// TIA Portal project "plc_logging_siemens" (V17)

(* hardware
DEVICE "S7-1500/ET200MP station_1"  S7-1500 station
   slot 0: "Rail_0"  Rack  6ES7 590-1***0-0AA0
   slot 1: "PLC_1"  CPU 1511T-1 PN  6ES7 511-1TK01-0AB0  V2.9
      slot 3: "CPU display_1"  6ES7591-1AA00-0AA0
      slot 32768: "PROFINET interface_1"  X1
         slot 32769: "Port_1"  X1 P1
         slot 32770: "Port_2"  X1 P2
      slot 34817: "Virtual CP interface port_1"  Virtual CP interface port  Virtual CP interface port
*)

// ===== PLC "PLC_1"  CPU 1511T-1 PN =====

VAR_GLOBAL   // PLC tag table "Default tag table"
   "System_Byte" AT %MB1 : Byte;
   "FirstScan" AT %M1.0 : Bool;
   "DiagStatusUpdate" AT %M1.1 : Bool;
   "AlwaysTRUE" AT %M1.2 : Bool;
   "AlwaysFALSE" AT %M1.3 : Bool;
   "Clock_Byte" AT %MB0 : Byte;
   "Clock_10Hz" AT %M0.0 : Bool;
   "Clock_5Hz" AT %M0.1 : Bool;
   "Clock_2.5Hz" AT %M0.2 : Bool;
   "Clock_2Hz" AT %M0.3 : Bool;
   "Clock_1.25Hz" AT %M0.4 : Bool;
   "Clock_1Hz" AT %M0.5 : Bool;
   "Clock_0.625Hz" AT %M0.6 : Bool;
   "Clock_0.5Hz" AT %M0.7 : Bool;
END_VAR

DATA_BLOCK "test_logger_DB"   // DB2
{ S7_Optimized_Access := 'TRUE' }
VERSION : 0.1
// stored: InstanceOfName test_logger
"test_logger"
BEGIN
END_DATA_BLOCK

// folder: logger

DATA_BLOCK "logger"   // DB1
{ S7_Optimized_Access := 'TRUE' }
VERSION : 0.1
// stored: InstanceOfName LoggerFb
"LoggerFb"
BEGIN
END_DATA_BLOCK

DATA_BLOCK "LoggerLevels"   // DB3
{ S7_Optimized_Access := 'TRUE' }
VERSION : 0.1
   VAR
      NOTSET : USInt := 0;   // logging everything
      DEBUG : USInt := 10;
      INFO : USInt := 20;
      WARNING : USInt := 30;
      ERROR : USInt := 40;
      CRITICAL : USInt := 50;
      DISABLE : USInt := 100;   // logging disabled
   END_VAR
BEGIN
END_DATA_BLOCK

// folder: (top level)

FUNCTION_BLOCK "test_logger"   // FB2, SCL
{ S7_Optimized_Access := 'TRUE' }
VERSION : 0.1
   VAR
      prev : Struct
         clock : Bool;
      END_STRUCT;
   END_VAR
BEGIN
   "logger.config_in_block"(level := "LoggerLevels".DEBUG,
                            block_title := 'test_logger_block');


   if "Clock_0.5Hz" AND NOT #prev.clock THEN
       "logger.debug_3"(msg := 'test debug message, SP: {0}, PV: {1}, add: {2}',
                        value_0 := REAL_TO_STRING(10),
                        value_1 := REAL_TO_STRING(11),
                        value_2 := REAL_TO_STRING(12)
       );
       //"logger.info_0"('test info message');
       //"logger.warning_0"('test warning message');
       //"logger.error_0"('test error message');
       //"logger.critical_0"(msg := 'test critical message');
   END_IF;

   #prev.clock := "Clock_0.5Hz";
END_FUNCTION_BLOCK

ORGANIZATION_BLOCK "Main"   // OB1, SCL, ProgramCycle
TITLE = "Main Program Sweep (Cycle)"
{ S7_Optimized_Access := 'TRUE' }
VERSION : 0.1
   VAR_INPUT
      Initial_Call : Bool;   // Initial call of this OB
      Remanence : Bool;   // =True, if remanent data are available
   END_VAR
BEGIN
   "test_logger_DB"();


   "logger"(global_logger_level := "LoggerLevels".DEBUG,
            ip_1 := 10,
            ip_2 := 101,
            ip_3 := 50,
            ip_4 := 17,
            port_number := 8000,
            interface_id := "Local~PROFINET_interface_1"
   );
END_ORGANIZATION_BLOCK

// folder: logger

FUNCTION_BLOCK "LoggerFb"   // FB1, SCL
{ S7_Optimized_Access := 'TRUE' }
VERSION : 0.1
   VAR_INPUT
      global_logger_level : USInt := 0;   // Filter all logging messages
      ip_1 : USInt := 192;
      ip_2 : USInt := 168;
      ip_3 : USInt := 10;
      ip_4 : USInt := 2;
      port_number : UInt := 4567;
      interface_id : UInt := 64;
   END_VAR
   VAR_OUTPUT
      buffer_size : Int;
   END_VAR
   VAR
      prev : Struct
         state : Int;
      END_STRUCT;
      diag : Struct
         tcon_done_counter : UDInt;
         tcon_error_counter : UDInt;
         tcon_error_status : Word;
         timeout_counter : UDInt;
         tsend_done_counter : UDInt;
         tsend_error_counter : UDInt;
         tsend_error_status : Word;
      END_STRUCT;
      connect : TCON_IP_v4;
      data : String;
      buffer : Array[0..9] of String;
      state : Int;
      timeout : TON_TIME;
      init : Bool := TRUE;   // TRUE = initialize function block
      config_in_block : Struct
         level : USInt;
         block_title : String;
      END_STRUCT;
      tcon : TCON;
      tsend : TSEND;
      tdiscon : TDISCON;
      connect_id : Conn_Ouc := 16#0001;
   END_VAR
   VAR_TEMP
      i : Int;
      com_rst : Bool;
   END_VAR
   VAR CONSTANT
      BUFFER_SIZE_ : Int := 9;
      ST_STOP : Int;
      ST_CONNECT : Int := 1;
      ST_WAIT : Int := 2;
      ST_SEND : Int := 3;
      ST_DISCON : Int := 4;
   END_VAR
BEGIN
   (*Блок логгера.*)

   // -----------------------------------------------------------------------------

   if #init THEN
       // first execution
       #connect.RemoteAddress.ADDR[1] := #ip_1;
       #connect.RemoteAddress.ADDR[2] := #ip_2;
       #connect.RemoteAddress.ADDR[3] := #ip_3;
       #connect.RemoteAddress.ADDR[4] := #ip_4;
       #connect.RemotePort := #port_number;
       #connect.LocalPort := #port_number;
       #connect.ActiveEstablished := true;
       #connect.InterfaceId := #interface_id;
       //#connect.ID := #id;
       #state := #ST_STOP;
       #connect.ConnectionType := 11;

       #buffer_size := #"BUFFER_SIZE_";
   END_IF;

   case #state OF
       #ST_STOP:
           if #global_logger_level < "LoggerLevels".DISABLE THEN
               #state := #ST_CONNECT;
               for #i := 0 TO #"BUFFER_SIZE_" DO
                   #buffer[#i] := '';
               END_FOR;
           END_IF;

       #ST_CONNECT:
           if #global_logger_level = "LoggerLevels".DISABLE OR #init THEN
               #state := #ST_STOP;
           ELSIF #tcon.DONE THEN
               // done
               #diag.tcon_done_counter += 1;
               #state := #ST_WAIT;
           ELSIF #tcon.ERROR THEN
               // error
               #diag.tcon_error_counter += 1;
               #diag.tcon_error_status := #tcon.STATUS;
               #state := #ST_STOP;
               if #tcon.STATUS = 16#80A3 THEN
                   #connect_id += 1;
               END_IF;
           ELSIF #timeout.Q THEN
               // timeout
               #diag.timeout_counter += 1;
               #state := #ST_STOP;
           END_IF;

       #ST_WAIT:
           if #global_logger_level = "LoggerLevels".DISABLE OR #init THEN
               #state := #ST_DISCON;
           END_IF;

           if #buffer[0] <> '' THEN
               #data := #buffer[0];
               for #i := 0 TO #"BUFFER_SIZE_" - 1 DO
                   #buffer[#i] := #buffer[#i + 1];
               END_FOR;
               #buffer[#"BUFFER_SIZE_"] := '';
               #state := #ST_SEND;
           END_IF;

       #ST_SEND:
           if #global_logger_level = "LoggerLevels".DISABLE OR #init THEN
               #state := #ST_DISCON;
           ELSIF #tsend.DONE THEN
               // done
               #diag.tsend_done_counter += 1;
               #state := #ST_WAIT;
           ELSIF #tsend.ERROR THEN
               // error
               #diag.tsend_error_counter += 1;
               #diag.tsend_error_status := #tsend.STATUS;
               #state := #ST_DISCON;
           ELSIF #timeout.Q THEN
               // timeout
               #diag.timeout_counter += 1;
               #state := #ST_DISCON;
           END_IF;

       #ST_DISCON:
           if #tdiscon.DONE OR #tdiscon.ERROR OR #timeout.Q THEN
               #state := #ST_STOP;
           END_IF;

   END_CASE;

   #timeout(IN := #state = #prev.state,
            PT := T#5s);

   #connect.ID := #connect_id;
   #tcon(REQ := #state = #ST_CONNECT,
         ID := #connect_id,
         CONNECT := #connect);

   #tsend(REQ := #state = #ST_SEND,
          ID := #connect_id,
          LEN := INT_TO_UDINT(LEN(#data)) + 2, // why 2 ???
          DATA := #data);

   #tdiscon(REQ := #state = #ST_DISCON,
            ID := #connect_id);

   #init := false;
   #prev.state := #state;
END_FUNCTION_BLOCK

FUNCTION "logger.debug_1" : Void   // FC1, SCL
{ S7_Optimized_Access := 'TRUE' }
VERSION : 0.1
   VAR_INPUT
      msg : String;   // message for logging
      value_0 : String;   // additional value 0
   END_VAR
   VAR_TEMP
      str : String;
   END_VAR
BEGIN
   IF MAX_USINT(IN1 := "logger".config_in_block.level, IN2 := "logger".global_logger_level) >
       "LoggerLevels".DEBUG THEN
       RETURN;
   END_IF;

   #str := '';
   #str := CONCAT_STRING(IN1 := #str, IN2 := #msg);
   #str := CONCAT_STRING(IN1 := #str, IN2 := '$t');
   #str := CONCAT_STRING(IN1 := #str, IN2 := #value_0);

   "logger._log"(level := "LoggerLevels".DEBUG,
                 msg := #str
   );
END_FUNCTION

FUNCTION "logger._log" : Void   // FC2, SCL
{ S7_Optimized_Access := 'TRUE' }
VERSION : 0.1
   VAR_INPUT
      level : USInt;
      msg : String;
   END_VAR
   VAR_TEMP
      temp_dtl : DTL;
      temp_int : Int;
      ts : String;
      pos : UInt;
      i : Int;
      str : String;
   END_VAR
BEGIN
   (*Add message to buffer.
   Format: LEVEL, TIMESTAMP, BLOCK_TITLE, MESSAGE
   Separator - \t.
   *)

   REGION timestamp
       // timestamp
       #temp_int := RD_LOC_T(#temp_dtl);

       #ts := 'YYYY-MM-DD HH:MM:SS,NNNNNNNNN';
       #pos := 1;
       VAL_STRG(IN := #temp_dtl.YEAR,
                SIZE := 4,
                PREC := 0,
                FORMAT := 0,
                P := #pos,
                OUT => #ts);
       #pos := 6;
       VAL_STRG(IN := #temp_dtl.MONTH,
                SIZE := 2,
                PREC := 0,
                FORMAT := 0,
                P := #pos,
                OUT => #ts);
       #pos := 9;
       VAL_STRG(IN := #temp_dtl.DAY,
                SIZE := 2,
                PREC := 0,
                FORMAT := 0,
                P := #pos,
                OUT => #ts);
       #pos := 12;
       VAL_STRG(IN := #temp_dtl.HOUR,
                SIZE := 2,
                PREC := 0,
                FORMAT := 0,
                P := #pos,
                OUT => #ts);
       #pos := 15;
       VAL_STRG(IN := #temp_dtl.MINUTE,
                SIZE := 2,
                PREC := 0,
                FORMAT := 0,
                P := #pos,
                OUT => #ts);
       #pos := 18;
       VAL_STRG(IN := #temp_dtl.SECOND,
                SIZE := 2,
                PREC := 0,
                FORMAT := 0,
                P := #pos,
                OUT => #ts);
       #pos := 21;
       VAL_STRG(IN := #temp_dtl.NANOSECOND,
                SIZE := 0,
                PREC := 0,
                FORMAT := 0,
                P := #pos,
                OUT => #ts);
       FOR #i := 1 TO LEN(#ts) DO
           // fill with zeros
           IF #ts[#i] = ' ' THEN
               #ts[#i] := '0';
           END_IF;
       END_FOR;
       #ts[11] := ' '; // separator between day and hours
   END_REGION

   #str := '';
   #str := CONCAT_STRING(IN1 := #str, IN2 := USINT_TO_STRING(#level));
   #str := CONCAT_STRING(IN1 := #str, IN2 := '$t');
   #str := CONCAT_STRING(IN1 := #str, IN2 := #ts);
   #str := CONCAT_STRING(IN1 := #str, IN2 := '$t');
   #str := CONCAT_STRING(IN1 := #str, IN2 := "logger".config_in_block.block_title);
   #str := CONCAT_STRING(IN1 := #str, IN2 := '$t');
   #str := CONCAT_STRING(IN1 := #str, IN2 := #msg);
   #str := CONCAT_STRING(IN1 := #str, IN2 := '$r');

   FOR #i := 0 TO "logger".buffer_size DO
       IF "logger".buffer[#i] = '' THEN
           "logger".buffer[#i] := #str;
           RETURN;
       END_IF;
   END_FOR;
END_FUNCTION

FUNCTION "logger.debug_0" : Void   // FC3, SCL
{ S7_Optimized_Access := 'TRUE' }
VERSION : 0.1
   VAR_INPUT
      msg : String;   // message for logging
   END_VAR
BEGIN
   IF MAX_USINT(IN1 := "logger".config_in_block.level, IN2 := "logger".global_logger_level) >
       "LoggerLevels".DEBUG THEN
       RETURN;
   END_IF;

   "logger._log"(level := "LoggerLevels".DEBUG,
                 msg := #msg
   );
END_FUNCTION

FUNCTION "logger.info_0" : Void   // FC4, SCL
{ S7_Optimized_Access := 'TRUE' }
VERSION : 0.1
   VAR_INPUT
      msg : String;   // message for logging
   END_VAR
BEGIN
   IF MAX_USINT(IN1 := "logger".config_in_block.level, IN2 := "logger".global_logger_level) >
       "LoggerLevels".INFO THEN
       RETURN;
   END_IF;

   "logger._log"(level := "LoggerLevels".INFO,
                 msg := #msg
   );
END_FUNCTION

FUNCTION "logger.config_in_block" : Void   // FC5, SCL
{ S7_Optimized_Access := 'TRUE' }
VERSION : 0.1
   VAR_INPUT
      level : USInt;
      block_title : String;
   END_VAR
BEGIN
   "logger".config_in_block.block_title := #block_title;
   "logger".config_in_block.level := #level;
END_FUNCTION

FUNCTION "logger.warning_0" : Void   // FC6, SCL
{ S7_Optimized_Access := 'TRUE' }
VERSION : 0.1
   VAR_INPUT
      msg : String;   // message for logging
   END_VAR
BEGIN
   IF MAX_USINT(IN1 := "logger".config_in_block.level, IN2 := "logger".global_logger_level) >
       "LoggerLevels".WARNING THEN
       RETURN;
   END_IF;

   "logger._log"(level := "LoggerLevels".WARNING,
                 msg := #msg
   );
END_FUNCTION

FUNCTION "logger.error_0" : Void   // FC7, SCL
{ S7_Optimized_Access := 'TRUE' }
VERSION : 0.1
   VAR_INPUT
      msg : String;   // message for logging
   END_VAR
BEGIN
   IF MAX_USINT(IN1 := "logger".config_in_block.level, IN2 := "logger".global_logger_level) >
       "LoggerLevels".ERROR THEN
       RETURN;
   END_IF;

   "logger._log"(level := "LoggerLevels".ERROR,
                 msg := #msg
   );
END_FUNCTION

FUNCTION "logger.critical_0" : Void   // FC8, SCL
{ S7_Optimized_Access := 'TRUE' }
VERSION : 0.1
   VAR_INPUT
      msg : String;   // message for logging
   END_VAR
BEGIN
   IF MAX_USINT(IN1 := "logger".config_in_block.level, IN2 := "logger".global_logger_level) >
       "LoggerLevels".CRITICAL THEN
       RETURN;
   END_IF;

   "logger._log"(level := "LoggerLevels".CRITICAL,
                 msg := #msg
   );
END_FUNCTION

FUNCTION "logger.debug_2" : Void   // FC9, SCL
{ S7_Optimized_Access := 'TRUE' }
VERSION : 0.1
   VAR_INPUT
      msg : String;   // message for logging
      value_0 : String;   // additional value 0
      value_1 : String;   // additional value 1
   END_VAR
   VAR_TEMP
      str : String;
   END_VAR
BEGIN
   IF MAX_USINT(IN1 := "logger".config_in_block.level, IN2 := "logger".global_logger_level) >
       "LoggerLevels".DEBUG THEN
       RETURN;
   END_IF;

   #str := '';
   #str := CONCAT_STRING(IN1 := #str, IN2 := #msg);
   #str := CONCAT_STRING(IN1 := #str, IN2 := '$t');
   #str := CONCAT_STRING(IN1 := #str, IN2 := #value_0);
   #str := CONCAT_STRING(IN1 := #str, IN2 := '$t');
   #str := CONCAT_STRING(IN1 := #str, IN2 := #value_1);

   "logger._log"(level := "LoggerLevels".DEBUG,
                 msg := #str
   );
END_FUNCTION

FUNCTION "logger.debug_3" : Void   // FC10, SCL
{ S7_Optimized_Access := 'TRUE' }
VERSION : 0.1
   VAR_INPUT
      msg : String;   // message for logging
      value_0 : String;   // additional value 0
      value_1 : String;   // additional value 1
      value_2 : String;   // additional value 2
   END_VAR
   VAR_TEMP
      str : String;
   END_VAR
BEGIN
   IF MAX_USINT(IN1 := "logger".config_in_block.level, IN2 := "logger".global_logger_level) >
       "LoggerLevels".DEBUG THEN
       RETURN;
   END_IF;

   #str := '';
   #str := CONCAT_STRING(IN1 := #str, IN2 := #msg);
   #str := CONCAT_STRING(IN1 := #str, IN2 := '$t');
   #str := CONCAT_STRING(IN1 := #str, IN2 := #value_0);
   #str := CONCAT_STRING(IN1 := #str, IN2 := '$t');
   #str := CONCAT_STRING(IN1 := #str, IN2 := #value_1);
   #str := CONCAT_STRING(IN1 := #str, IN2 := '$t');
   #str := CONCAT_STRING(IN1 := #str, IN2 := #value_2);

   "logger._log"(level := "LoggerLevels".DEBUG,
                 msg := #str
   );
END_FUNCTION

FUNCTION "logger.info_1" : Void   // FC11, SCL
{ S7_Optimized_Access := 'TRUE' }
VERSION : 0.1
   VAR_INPUT
      msg : String;   // message for logging
      value_0 : String;   // additional value 0
   END_VAR
   VAR_TEMP
      str : String;
   END_VAR
BEGIN
   IF MAX_USINT(IN1 := "logger".config_in_block.level, IN2 := "logger".global_logger_level) >
       "LoggerLevels".INFO THEN
       RETURN;
   END_IF;

   #str := '';
   #str := CONCAT_STRING(IN1 := #str, IN2 := #msg);
   #str := CONCAT_STRING(IN1 := #str, IN2 := '$t');
   #str := CONCAT_STRING(IN1 := #str, IN2 := #value_0);

   "logger._log"(level := "LoggerLevels".INFO,
                 msg := #str
   );
END_FUNCTION

FUNCTION "logger.error_1" : Void   // FC12, SCL
{ S7_Optimized_Access := 'TRUE' }
VERSION : 0.1
   VAR_INPUT
      msg : String;   // message for logging
      value_0 : String;   // additional value 0
   END_VAR
   VAR_TEMP
      str : String;
   END_VAR
BEGIN
   IF MAX_USINT(IN1 := "logger".config_in_block.level, IN2 := "logger".global_logger_level) >
       "LoggerLevels".ERROR THEN
       RETURN;
   END_IF;

   #str := '';
   #str := CONCAT_STRING(IN1 := #str, IN2 := #msg);
   #str := CONCAT_STRING(IN1 := #str, IN2 := '$t');
   #str := CONCAT_STRING(IN1 := #str, IN2 := #value_0);

   "logger._log"(level := "LoggerLevels".ERROR,
                 msg := #str
   );
END_FUNCTION

FUNCTION "logger.critical_1" : Void   // FC13, SCL
{ S7_Optimized_Access := 'TRUE' }
VERSION : 0.1
   VAR_INPUT
      msg : String;   // message for logging
      value_0 : String;   // additional value 0
   END_VAR
   VAR_TEMP
      str : String;
   END_VAR
BEGIN
   IF MAX_USINT(IN1 := "logger".config_in_block.level, IN2 := "logger".global_logger_level) >
       "LoggerLevels".CRITICAL THEN
       RETURN;
   END_IF;

   #str := '';
   #str := CONCAT_STRING(IN1 := #str, IN2 := #msg);
   #str := CONCAT_STRING(IN1 := #str, IN2 := '$t');
   #str := CONCAT_STRING(IN1 := #str, IN2 := #value_0);

   "logger._log"(level := "LoggerLevels".CRITICAL,
                 msg := #str
   );
END_FUNCTION

FUNCTION "logger.warning_1" : Void   // FC14, SCL
{ S7_Optimized_Access := 'TRUE' }
VERSION : 0.1
   VAR_INPUT
      msg : String;   // message for logging
      value_0 : String;   // additional value 0
   END_VAR
   VAR_TEMP
      str : String;
   END_VAR
BEGIN
   IF MAX_USINT(IN1 := "logger".config_in_block.level, IN2 := "logger".global_logger_level) >
       "LoggerLevels".WARNING THEN
       RETURN;
   END_IF;

   #str := '';
   #str := CONCAT_STRING(IN1 := #str, IN2 := #msg);
   #str := CONCAT_STRING(IN1 := #str, IN2 := '$t');
   #str := CONCAT_STRING(IN1 := #str, IN2 := #value_0);

   "logger._log"(level := "LoggerLevels".WARNING,
                 msg := #str
   );
END_FUNCTION

FUNCTION "logger.warning_2" : Void   // FC15, SCL
{ S7_Optimized_Access := 'TRUE' }
VERSION : 0.1
   VAR_INPUT
      msg : String;   // message for logging
      value_0 : String;   // additional value 0
      value_1 : String;   // additional value 1
   END_VAR
   VAR_TEMP
      str : String;
   END_VAR
BEGIN
   IF MAX_USINT(IN1 := "logger".config_in_block.level, IN2 := "logger".global_logger_level) >
       "LoggerLevels".WARNING THEN
       RETURN;
   END_IF;

   #str := '';
   #str := CONCAT_STRING(IN1 := #str, IN2 := #msg);
   #str := CONCAT_STRING(IN1 := #str, IN2 := '$t');
   #str := CONCAT_STRING(IN1 := #str, IN2 := #value_0);
   #str := CONCAT_STRING(IN1 := #str, IN2 := '$t');
   #str := CONCAT_STRING(IN1 := #str, IN2 := #value_1);

   "logger._log"(level := "LoggerLevels".WARNING,
                 msg := #str
   );
END_FUNCTION

FUNCTION "logger.info_2" : Void   // FC16, SCL
{ S7_Optimized_Access := 'TRUE' }
VERSION : 0.1
   VAR_INPUT
      msg : String;   // message for logging
      value_0 : String;   // additional value 0
      value_1 : String;   // additional value 1
   END_VAR
   VAR_TEMP
      str : String;
   END_VAR
BEGIN
   IF MAX_USINT(IN1 := "logger".config_in_block.level, IN2 := "logger".global_logger_level) >
       "LoggerLevels".INFO THEN
       RETURN;
   END_IF;

   #str := '';
   #str := CONCAT_STRING(IN1 := #str, IN2 := #msg);
   #str := CONCAT_STRING(IN1 := #str, IN2 := '$t');
   #str := CONCAT_STRING(IN1 := #str, IN2 := #value_0);
   #str := CONCAT_STRING(IN1 := #str, IN2 := '$t');
   #str := CONCAT_STRING(IN1 := #str, IN2 := #value_1);

   "logger._log"(level := "LoggerLevels".INFO,
                 msg := #str
   );
END_FUNCTION

FUNCTION "logger.critical_2" : Void   // FC17, SCL
{ S7_Optimized_Access := 'TRUE' }
VERSION : 0.1
   VAR_INPUT
      msg : String;   // message for logging
      value_0 : String;   // additional value 0
      value_1 : String;   // additional value 1
   END_VAR
   VAR_TEMP
      str : String;
   END_VAR
BEGIN
   IF MAX_USINT(IN1 := "logger".config_in_block.level, IN2 := "logger".global_logger_level) >
       "LoggerLevels".CRITICAL THEN
       RETURN;
   END_IF;

   #str := '';
   #str := CONCAT_STRING(IN1 := #str, IN2 := #msg);
   #str := CONCAT_STRING(IN1 := #str, IN2 := '$t');
   #str := CONCAT_STRING(IN1 := #str, IN2 := #value_0);
   #str := CONCAT_STRING(IN1 := #str, IN2 := '$t');
   #str := CONCAT_STRING(IN1 := #str, IN2 := #value_1);

   "logger._log"(level := "LoggerLevels".CRITICAL,
                 msg := #str
   );
END_FUNCTION

FUNCTION "logger.error_2" : Void   // FC18, SCL
{ S7_Optimized_Access := 'TRUE' }
VERSION : 0.1
   VAR_INPUT
      msg : String;   // message for logging
      value_0 : String;   // additional value 0
      value_1 : String;   // additional value 1
   END_VAR
   VAR_TEMP
      str : String;
   END_VAR
BEGIN
   IF MAX_USINT(IN1 := "logger".config_in_block.level, IN2 := "logger".global_logger_level) >
       "LoggerLevels".ERROR THEN
       RETURN;
   END_IF;

   #str := '';
   #str := CONCAT_STRING(IN1 := #str, IN2 := #msg);
   #str := CONCAT_STRING(IN1 := #str, IN2 := '$t');
   #str := CONCAT_STRING(IN1 := #str, IN2 := #value_0);
   #str := CONCAT_STRING(IN1 := #str, IN2 := '$t');
   #str := CONCAT_STRING(IN1 := #str, IN2 := #value_1);

   "logger._log"(level := "LoggerLevels".ERROR,
                 msg := #str
   );
END_FUNCTION

FUNCTION "logger.error_3" : Void   // FC19, SCL
{ S7_Optimized_Access := 'TRUE' }
VERSION : 0.1
   VAR_INPUT
      msg : String;   // message for logging
      value_0 : String;   // additional value 0
      value_1 : String;   // additional value 1
      value_2 : String;   // additional value 2
   END_VAR
   VAR_TEMP
      str : String;
   END_VAR
BEGIN
   IF MAX_USINT(IN1 := "logger".config_in_block.level, IN2 := "logger".global_logger_level) >
       "LoggerLevels".ERROR THEN
       RETURN;
   END_IF;

   #str := '';
   #str := CONCAT_STRING(IN1 := #str, IN2 := #msg);
   #str := CONCAT_STRING(IN1 := #str, IN2 := '$t');
   #str := CONCAT_STRING(IN1 := #str, IN2 := #value_0);
   #str := CONCAT_STRING(IN1 := #str, IN2 := '$t');
   #str := CONCAT_STRING(IN1 := #str, IN2 := #value_1);
   #str := CONCAT_STRING(IN1 := #str, IN2 := '$t');
   #str := CONCAT_STRING(IN1 := #str, IN2 := #value_2);

   "logger._log"(level := "LoggerLevels".ERROR,
                 msg := #str
   );
END_FUNCTION

FUNCTION "logger.info_3" : Void   // FC20, SCL
{ S7_Optimized_Access := 'TRUE' }
VERSION : 0.1
   VAR_INPUT
      msg : String;   // message for logging
      value_0 : String;   // additional value 0
      value_1 : String;   // additional value 1
      value_2 : String;   // additional value 2
   END_VAR
   VAR_TEMP
      str : String;
   END_VAR
BEGIN
   IF MAX_USINT(IN1 := "logger".config_in_block.level, IN2 := "logger".global_logger_level) >
       "LoggerLevels".INFO THEN
       RETURN;
   END_IF;

   #str := '';
   #str := CONCAT_STRING(IN1 := #str, IN2 := #msg);
   #str := CONCAT_STRING(IN1 := #str, IN2 := '$t');
   #str := CONCAT_STRING(IN1 := #str, IN2 := #value_0);
   #str := CONCAT_STRING(IN1 := #str, IN2 := '$t');
   #str := CONCAT_STRING(IN1 := #str, IN2 := #value_1);
   #str := CONCAT_STRING(IN1 := #str, IN2 := '$t');
   #str := CONCAT_STRING(IN1 := #str, IN2 := #value_2);

   "logger._log"(level := "LoggerLevels".INFO,
                 msg := #str
   );
END_FUNCTION

FUNCTION "logger.critical_3" : Void   // FC21, SCL
{ S7_Optimized_Access := 'TRUE' }
VERSION : 0.1
   VAR_INPUT
      msg : String;   // message for logging
      value_0 : String;   // additional value 0
      value_1 : String;   // additional value 1
      value_2 : String;   // additional value 2
   END_VAR
   VAR_TEMP
      str : String;
   END_VAR
BEGIN
   IF MAX_USINT(IN1 := "logger".config_in_block.level, IN2 := "logger".global_logger_level) >
       "LoggerLevels".CRITICAL THEN
       RETURN;
   END_IF;

   #str := '';
   #str := CONCAT_STRING(IN1 := #str, IN2 := #msg);
   #str := CONCAT_STRING(IN1 := #str, IN2 := '$t');
   #str := CONCAT_STRING(IN1 := #str, IN2 := #value_0);
   #str := CONCAT_STRING(IN1 := #str, IN2 := '$t');
   #str := CONCAT_STRING(IN1 := #str, IN2 := #value_1);
   #str := CONCAT_STRING(IN1 := #str, IN2 := '$t');
   #str := CONCAT_STRING(IN1 := #str, IN2 := #value_2);

   "logger._log"(level := "LoggerLevels".CRITICAL,
                 msg := #str
   );
END_FUNCTION

FUNCTION "logger.warning_3" : Void   // FC22, SCL
{ S7_Optimized_Access := 'TRUE' }
VERSION : 0.1
   VAR_INPUT
      msg : String;   // message for logging
      value_0 : String;   // additional value 0
      value_1 : String;   // additional value 1
      value_2 : String;   // additional value 2
   END_VAR
   VAR_TEMP
      str : String;
   END_VAR
BEGIN
   IF MAX_USINT(IN1 := "logger".config_in_block.level, IN2 := "logger".global_logger_level) >
       "LoggerLevels".WARNING THEN
       RETURN;
   END_IF;

   #str := '';
   #str := CONCAT_STRING(IN1 := #str, IN2 := #msg);
   #str := CONCAT_STRING(IN1 := #str, IN2 := '$t');
   #str := CONCAT_STRING(IN1 := #str, IN2 := #value_0);
   #str := CONCAT_STRING(IN1 := #str, IN2 := '$t');
   #str := CONCAT_STRING(IN1 := #str, IN2 := #value_1);
   #str := CONCAT_STRING(IN1 := #str, IN2 := '$t');
   #str := CONCAT_STRING(IN1 := #str, IN2 := #value_2);

   "logger._log"(level := "LoggerLevels".WARNING,
                 msg := #str
   );
END_FUNCTION

// ===== library: MasterCopy "Copy of Program blocks in logger" =====

// folder: logger

DATA_BLOCK "logger"   // DB1
{ S7_Optimized_Access := 'TRUE' }
VERSION : 0.1
// stored: InstanceOfName LoggerFb
"LoggerFb"
BEGIN
END_DATA_BLOCK

DATA_BLOCK "LoggerLevels"   // DB3
{ S7_Optimized_Access := 'TRUE' }
VERSION : 0.1
   VAR
      NOTSET : USInt := 0;   // logging everything
      DEBUG : USInt := 10;
      INFO : USInt := 20;
      WARNING : USInt := 30;
      ERROR : USInt := 40;
      CRITICAL : USInt := 50;
      DISABLE : USInt := 100;   // logging disabled
   END_VAR
BEGIN
END_DATA_BLOCK

FUNCTION_BLOCK "LoggerFb"   // FB1, SCL
{ S7_Optimized_Access := 'TRUE' }
VERSION : 0.1
   VAR_INPUT
      global_logger_level : USInt := 0;   // Filter all logging messages
      ip_1 : USInt := 10;
      ip_2 : USInt := 101;
      ip_3 : USInt := 50;
      ip_4 : USInt := 17;
      port_number : UInt := 4567;
      interface_id : UInt := 64;
      id : Conn_Ouc := 1;
   END_VAR
   VAR_OUTPUT
      buffer_size : Int;
   END_VAR
   VAR
      tsend : TSEND_C;
      connect : TCON_IP_v4;
      data : String;
      buffer : Array[0..9] of String;
      state : Int;
      timeout : TON_TIME;
      init : Bool := TRUE;   // TRUE = initialize function block
      config_in_block : Struct
         level : USInt;
         block_title : String;
      END_STRUCT;
   END_VAR
   VAR_TEMP
      i : Int;
   END_VAR
   VAR CONSTANT
      ST_STOP : Int;
      ST_WAIT : Int := 1;
      ST_SEND : Int := 2;
      BUFFER_SIZE_ : Int := 9;
   END_VAR
BEGIN
   (*Блок логгера.*)

   // -----------------------------------------------------------------------------

   if #init THEN
       // first execution
       #init := false;
       #connect.RemoteAddress.ADDR[1] := #ip_1;
       #connect.RemoteAddress.ADDR[2] := #ip_2;
       #connect.RemoteAddress.ADDR[3] := #ip_3;
       #connect.RemoteAddress.ADDR[4] := #ip_4;
       #connect.RemotePort := #port_number;
       #connect.LocalPort := #port_number;
       #connect.ActiveEstablished := true;
       #connect.InterfaceId := #interface_id;
       #connect.ID := #id;
       #state := #ST_STOP;
       #connect.ConnectionType := 11;

       #buffer_size := #"BUFFER_SIZE_";
   END_IF;


   case #state OF
       #ST_STOP:
           if #global_logger_level < "LoggerLevels".DISABLE THEN
               #state := #ST_WAIT;
               for #i := 0 TO #"BUFFER_SIZE_" DO
                   #buffer[#i] := '';
               END_FOR;
           END_IF;

       #ST_WAIT:
           if #global_logger_level = "LoggerLevels".DISABLE THEN
               #state := #ST_STOP;
           END_IF;

           if #buffer[0] <> '' THEN
               #data := #buffer[0];
               for #i := 0 TO #"BUFFER_SIZE_" - 1 DO
                   #buffer[#i] := #buffer[#i + 1];
               END_FOR;
               #buffer[#"BUFFER_SIZE_"] := '';
               #state := #ST_SEND;
           END_IF;

       #ST_SEND:
           if #global_logger_level = "LoggerLevels".DISABLE THEN
               #state := #ST_STOP;
           ELSIF #tsend.DONE OR #tsend.ERROR OR #timeout.Q THEN
               #data := '';
               #state := #ST_WAIT;
           END_IF;

   END_CASE;

   #timeout(IN := #state = #ST_SEND,
            PT := T#30s);


   #tsend(REQ := #state = #ST_SEND,
          CONT := #state = #ST_SEND,
          CONNECT := #connect,
          DATA := #data
   );
END_FUNCTION_BLOCK

FUNCTION "logger.debug_1" : Void   // FC1, SCL
{ S7_Optimized_Access := 'TRUE' }
VERSION : 0.1
   VAR_INPUT
      msg : String;   // message for logging
      value_0 : String;   // additional value 0
   END_VAR
   VAR_TEMP
      str : String;
   END_VAR
BEGIN
   if "logger".config_in_block.level > "LoggerLevels".DEBUG THEN
       return;
   END_IF;

   #str := '';
   #str := CONCAT_STRING(IN1 := #str, IN2 := #msg);
   #str := CONCAT_STRING(IN1 := #str, IN2 := '$t');
   #str := CONCAT_STRING(IN1 := #str, IN2 := #value_0);

   "logger._log"(level := "LoggerLevels".DEBUG,
                 msg := #str
   );
END_FUNCTION

FUNCTION "logger._log" : Void   // FC2, SCL
{ S7_Optimized_Access := 'TRUE' }
VERSION : 0.1
   VAR_INPUT
      level : USInt;
      msg : String;
   END_VAR
   VAR_TEMP
      temp_dtl : DTL;
      temp_int : Int;
      ts : String;
      pos : UInt;
      i : Int;
      str : String;
   END_VAR
BEGIN
   (*Add message to buffer.
   Format: LEVEL, TIMESTAMP, BLOCK_TITLE, MESSAGE
   Separator - \t.
   *)

   region timestamp
       // timestamp
       #temp_int := RD_LOC_T(#temp_dtl);

       #ts := 'YYYY-MM-DD HH:MM:SS,NNNNNNNNN';
       #pos := 1;
       VAL_STRG(IN := #temp_dtl.YEAR,
                SIZE := 4,
                PREC := 0,
                FORMAT := 0,
                P := #pos,
                OUT => #ts);
       #pos := 6;
       VAL_STRG(IN := #temp_dtl.MONTH,
                SIZE := 2,
                PREC := 0,
                FORMAT := 0,
                P := #pos,
                OUT => #ts);
       #pos := 9;
       VAL_STRG(IN := #temp_dtl.DAY,
                SIZE := 2,
                PREC := 0,
                FORMAT := 0,
                P := #pos,
                OUT => #ts);
       #pos := 12;
       VAL_STRG(IN := #temp_dtl.HOUR,
                SIZE := 2,
                PREC := 0,
                FORMAT := 0,
                P := #pos,
                OUT => #ts);
       #pos := 15;
       VAL_STRG(IN := #temp_dtl.MINUTE,
                SIZE := 2,
                PREC := 0,
                FORMAT := 0,
                P := #pos,
                OUT => #ts);
       #pos := 18;
       VAL_STRG(IN := #temp_dtl.SECOND,
                SIZE := 2,
                PREC := 0,
                FORMAT := 0,
                P := #pos,
                OUT => #ts);
       #pos := 21;
       VAL_STRG(IN := #temp_dtl.NANOSECOND,
                SIZE := 0,
                PREC := 0,
                FORMAT := 0,
                P := #pos,
                OUT => #ts);
       for #i := 1 TO LEN(#ts) DO
           // fill with zeros
           if #ts[#i] = ' ' THEN
               #ts[#i] := '0';
           END_IF;
       END_FOR;
       #ts[11] := ' '; // separator between day and hours
   END_REGION

   #str := '';
   #str := CONCAT_STRING(IN1 := #str, IN2 := USINT_TO_STRING(#level));
   #str := CONCAT_STRING(IN1 := #str, IN2 := '$t');
   #str := CONCAT_STRING(IN1 := #str, IN2 := #ts);
   #str := CONCAT_STRING(IN1 := #str, IN2 := '$t');
   #str := CONCAT_STRING(IN1 := #str, IN2 := "logger".config_in_block.block_title);
   #str := CONCAT_STRING(IN1 := #str, IN2 := '$t');
   #str := CONCAT_STRING(IN1 := #str, IN2 := #msg);

   for #i := 0 TO "logger".buffer_size DO
       if "logger".buffer[#i] = '' THEN
           "logger".buffer[#i] := #str;
           return;
       END_IF;
   END_FOR;
END_FUNCTION

FUNCTION "logger.debug_0" : Void   // FC3, SCL
{ S7_Optimized_Access := 'TRUE' }
VERSION : 0.1
   VAR_INPUT
      msg : String;   // message for logging
   END_VAR
BEGIN

   if "logger".config_in_block.level > "LoggerLevels".DEBUG THEN
       return;
   END_IF;

   "logger._log"(level := "LoggerLevels".DEBUG,
                 msg := #msg
   );
END_FUNCTION

FUNCTION "logger.info_0" : Void   // FC4, SCL
{ S7_Optimized_Access := 'TRUE' }
VERSION : 0.1
   VAR_INPUT
      msg : String;   // message for logging
   END_VAR
BEGIN
   if "logger".config_in_block.level > "LoggerLevels".INFO THEN
       return;
   END_IF;

   "logger._log"(level := "LoggerLevels".INFO,
                 msg := #msg
   );
END_FUNCTION

FUNCTION "logger.config_in_block" : Void   // FC5, SCL
{ S7_Optimized_Access := 'TRUE' }
VERSION : 0.1
   VAR_INPUT
      level : USInt;
      block_title : String;
   END_VAR
BEGIN
   "logger".config_in_block.block_title := #block_title;
   "logger".config_in_block.level := #level;
END_FUNCTION

FUNCTION "logger.warning_0" : Void   // FC6, SCL
{ S7_Optimized_Access := 'TRUE' }
VERSION : 0.1
   VAR_INPUT
      msg : String;   // message for logging
   END_VAR
BEGIN
   if "logger".config_in_block.level > "LoggerLevels".WARNING THEN
       return;
   END_IF;

   "logger._log"(level := "LoggerLevels".WARNING,
                 msg := #msg
   );
END_FUNCTION

FUNCTION "logger.error_0" : Void   // FC7, SCL
{ S7_Optimized_Access := 'TRUE' }
VERSION : 0.1
   VAR_INPUT
      msg : String;   // message for logging
   END_VAR
BEGIN
   if "logger".config_in_block.level > "LoggerLevels".ERROR THEN
       return;
   END_IF;

   "logger._log"(level := "LoggerLevels".ERROR,
                 msg := #msg
   );
END_FUNCTION

FUNCTION "logger.critical_0" : Void   // FC8, SCL
{ S7_Optimized_Access := 'TRUE' }
VERSION : 0.1
   VAR_INPUT
      msg : String;   // message for logging
   END_VAR
BEGIN
   if "logger".config_in_block.level > "LoggerLevels".CRITICAL THEN
       return;
   END_IF;

   "logger._log"(level := "LoggerLevels".CRITICAL,
                 msg := #msg
   );
END_FUNCTION

FUNCTION "logger.debug_2" : Void   // FC9, SCL
{ S7_Optimized_Access := 'TRUE' }
VERSION : 0.1
   VAR_INPUT
      msg : String;   // message for logging
      value_0 : String;   // additional value 0
      value_1 : String;   // additional value 1
   END_VAR
   VAR_TEMP
      str : String;
   END_VAR
BEGIN
   if "logger".config_in_block.level > "LoggerLevels".DEBUG THEN
       return;
   END_IF;

   #str := '';
   #str := CONCAT_STRING(IN1 := #str, IN2 := #msg);
   #str := CONCAT_STRING(IN1 := #str, IN2 := '$t');
   #str := CONCAT_STRING(IN1 := #str, IN2 := #value_0);
   #str := CONCAT_STRING(IN1 := #str, IN2 := '$t');
   #str := CONCAT_STRING(IN1 := #str, IN2 := #value_1);

   "logger._log"(level := "LoggerLevels".DEBUG,
                 msg := #str
   );
END_FUNCTION

FUNCTION "logger.debug_3" : Void   // FC10, SCL
{ S7_Optimized_Access := 'TRUE' }
VERSION : 0.1
   VAR_INPUT
      msg : String;   // message for logging
      value_0 : String;   // additional value 0
      value_1 : String;   // additional value 1
      value_2 : String;   // additional value 2
   END_VAR
   VAR_TEMP
      str : String;
   END_VAR
BEGIN
   if "logger".config_in_block.level > "LoggerLevels".DEBUG THEN
       return;
   END_IF;

   #str := '';
   #str := CONCAT_STRING(IN1 := #str, IN2 := #msg);
   #str := CONCAT_STRING(IN1 := #str, IN2 := '$t');
   #str := CONCAT_STRING(IN1 := #str, IN2 := #value_0);
   #str := CONCAT_STRING(IN1 := #str, IN2 := '$t');
   #str := CONCAT_STRING(IN1 := #str, IN2 := #value_1);
   #str := CONCAT_STRING(IN1 := #str, IN2 := '$t');
   #str := CONCAT_STRING(IN1 := #str, IN2 := #value_2);

   "logger._log"(level := "LoggerLevels".DEBUG,
                 msg := #str
   );
END_FUNCTION

FUNCTION "logger.info_1" : Void   // FC11, SCL
{ S7_Optimized_Access := 'TRUE' }
VERSION : 0.1
   VAR_INPUT
      msg : String;   // message for logging
      value_0 : String;   // additional value 0
   END_VAR
   VAR_TEMP
      str : String;
   END_VAR
BEGIN
   if "logger".config_in_block.level > "LoggerLevels".INFO THEN
       return;
   END_IF;

   #str := '';
   #str := CONCAT_STRING(IN1 := #str, IN2 := #msg);
   #str := CONCAT_STRING(IN1 := #str, IN2 := '$t');
   #str := CONCAT_STRING(IN1 := #str, IN2 := #value_0);

   "logger._log"(level := "LoggerLevels".INFO,
                 msg := #str
   );
END_FUNCTION

FUNCTION "logger.error_1" : Void   // FC12, SCL
{ S7_Optimized_Access := 'TRUE' }
VERSION : 0.1
   VAR_INPUT
      msg : String;   // message for logging
      value_0 : String;   // additional value 0
   END_VAR
   VAR_TEMP
      str : String;
   END_VAR
BEGIN
   if "logger".config_in_block.level > "LoggerLevels".ERROR THEN
       return;
   END_IF;

   #str := '';
   #str := CONCAT_STRING(IN1 := #str, IN2 := #msg);
   #str := CONCAT_STRING(IN1 := #str, IN2 := '$t');
   #str := CONCAT_STRING(IN1 := #str, IN2 := #value_0);

   "logger._log"(level := "LoggerLevels".ERROR,
                 msg := #str
   );
END_FUNCTION

FUNCTION "logger.critical_1" : Void   // FC13, SCL
{ S7_Optimized_Access := 'TRUE' }
VERSION : 0.1
   VAR_INPUT
      msg : String;   // message for logging
      value_0 : String;   // additional value 0
   END_VAR
   VAR_TEMP
      str : String;
   END_VAR
BEGIN
   if "logger".config_in_block.level > "LoggerLevels".CRITICAL THEN
       return;
   END_IF;

   #str := '';
   #str := CONCAT_STRING(IN1 := #str, IN2 := #msg);
   #str := CONCAT_STRING(IN1 := #str, IN2 := '$t');
   #str := CONCAT_STRING(IN1 := #str, IN2 := #value_0);

   "logger._log"(level := "LoggerLevels".CRITICAL,
                 msg := #str
   );
END_FUNCTION

FUNCTION "logger.warning_1" : Void   // FC14, SCL
{ S7_Optimized_Access := 'TRUE' }
VERSION : 0.1
   VAR_INPUT
      msg : String;   // message for logging
      value_0 : String;   // additional value 0
   END_VAR
   VAR_TEMP
      str : String;
   END_VAR
BEGIN
   if "logger".config_in_block.level > "LoggerLevels".WARNING THEN
       return;
   END_IF;

   #str := '';
   #str := CONCAT_STRING(IN1 := #str, IN2 := #msg);
   #str := CONCAT_STRING(IN1 := #str, IN2 := '$t');
   #str := CONCAT_STRING(IN1 := #str, IN2 := #value_0);

   "logger._log"(level := "LoggerLevels".WARNING,
                 msg := #str
   );
END_FUNCTION

FUNCTION "logger.warning_2" : Void   // FC15, SCL
{ S7_Optimized_Access := 'TRUE' }
VERSION : 0.1
   VAR_INPUT
      msg : String;   // message for logging
      value_0 : String;   // additional value 0
      value_1 : String;   // additional value 1
   END_VAR
   VAR_TEMP
      str : String;
   END_VAR
BEGIN
   if "logger".config_in_block.level > "LoggerLevels".WARNING THEN
       return;
   END_IF;

   #str := '';
   #str := CONCAT_STRING(IN1 := #str, IN2 := #msg);
   #str := CONCAT_STRING(IN1 := #str, IN2 := '$t');
   #str := CONCAT_STRING(IN1 := #str, IN2 := #value_0);
   #str := CONCAT_STRING(IN1 := #str, IN2 := '$t');
   #str := CONCAT_STRING(IN1 := #str, IN2 := #value_1);

   "logger._log"(level := "LoggerLevels".WARNING,
                 msg := #str
   );
END_FUNCTION

FUNCTION "logger.info_2" : Void   // FC16, SCL
{ S7_Optimized_Access := 'TRUE' }
VERSION : 0.1
   VAR_INPUT
      msg : String;   // message for logging
      value_0 : String;   // additional value 0
      value_1 : String;   // additional value 1
   END_VAR
   VAR_TEMP
      str : String;
   END_VAR
BEGIN
   if "logger".config_in_block.level > "LoggerLevels".INFO THEN
       return;
   END_IF;

   #str := '';
   #str := CONCAT_STRING(IN1 := #str, IN2 := #msg);
   #str := CONCAT_STRING(IN1 := #str, IN2 := '$t');
   #str := CONCAT_STRING(IN1 := #str, IN2 := #value_0);
   #str := CONCAT_STRING(IN1 := #str, IN2 := '$t');
   #str := CONCAT_STRING(IN1 := #str, IN2 := #value_1);

   "logger._log"(level := "LoggerLevels".INFO,
                 msg := #str
   );
END_FUNCTION

FUNCTION "logger.critical_2" : Void   // FC17, SCL
{ S7_Optimized_Access := 'TRUE' }
VERSION : 0.1
   VAR_INPUT
      msg : String;   // message for logging
      value_0 : String;   // additional value 0
      value_1 : String;   // additional value 1
   END_VAR
   VAR_TEMP
      str : String;
   END_VAR
BEGIN
   if "logger".config_in_block.level > "LoggerLevels".CRITICAL THEN
       return;
   END_IF;

   #str := '';
   #str := CONCAT_STRING(IN1 := #str, IN2 := #msg);
   #str := CONCAT_STRING(IN1 := #str, IN2 := '$t');
   #str := CONCAT_STRING(IN1 := #str, IN2 := #value_0);
   #str := CONCAT_STRING(IN1 := #str, IN2 := '$t');
   #str := CONCAT_STRING(IN1 := #str, IN2 := #value_1);

   "logger._log"(level := "LoggerLevels".CRITICAL,
                 msg := #str
   );
END_FUNCTION

FUNCTION "logger.error_2" : Void   // FC18, SCL
{ S7_Optimized_Access := 'TRUE' }
VERSION : 0.1
   VAR_INPUT
      msg : String;   // message for logging
      value_0 : String;   // additional value 0
      value_1 : String;   // additional value 1
   END_VAR
   VAR_TEMP
      str : String;
   END_VAR
BEGIN
   if "logger".config_in_block.level > "LoggerLevels".ERROR THEN
       return;
   END_IF;

   #str := '';
   #str := CONCAT_STRING(IN1 := #str, IN2 := #msg);
   #str := CONCAT_STRING(IN1 := #str, IN2 := '$t');
   #str := CONCAT_STRING(IN1 := #str, IN2 := #value_0);
   #str := CONCAT_STRING(IN1 := #str, IN2 := '$t');
   #str := CONCAT_STRING(IN1 := #str, IN2 := #value_1);

   "logger._log"(level := "LoggerLevels".ERROR,
                 msg := #str
   );
END_FUNCTION

FUNCTION "logger.error_3" : Void   // FC19, SCL
{ S7_Optimized_Access := 'TRUE' }
VERSION : 0.1
   VAR_INPUT
      msg : String;   // message for logging
      value_0 : String;   // additional value 0
      value_1 : String;   // additional value 1
      value_2 : String;   // additional value 2
   END_VAR
   VAR_TEMP
      str : String;
   END_VAR
BEGIN
   if "logger".config_in_block.level > "LoggerLevels".ERROR THEN
       return;
   END_IF;

   #str := '';
   #str := CONCAT_STRING(IN1 := #str, IN2 := #msg);
   #str := CONCAT_STRING(IN1 := #str, IN2 := '$t');
   #str := CONCAT_STRING(IN1 := #str, IN2 := #value_0);
   #str := CONCAT_STRING(IN1 := #str, IN2 := '$t');
   #str := CONCAT_STRING(IN1 := #str, IN2 := #value_1);
   #str := CONCAT_STRING(IN1 := #str, IN2 := '$t');
   #str := CONCAT_STRING(IN1 := #str, IN2 := #value_2);

   "logger._log"(level := "LoggerLevels".ERROR,
                 msg := #str
   );
END_FUNCTION

FUNCTION "logger.info_3" : Void   // FC20, SCL
{ S7_Optimized_Access := 'TRUE' }
VERSION : 0.1
   VAR_INPUT
      msg : String;   // message for logging
      value_0 : String;   // additional value 0
      value_1 : String;   // additional value 1
      value_2 : String;   // additional value 2
   END_VAR
   VAR_TEMP
      str : String;
   END_VAR
BEGIN
   if "logger".config_in_block.level > "LoggerLevels".INFO THEN
       return;
   END_IF;

   #str := '';
   #str := CONCAT_STRING(IN1 := #str, IN2 := #msg);
   #str := CONCAT_STRING(IN1 := #str, IN2 := '$t');
   #str := CONCAT_STRING(IN1 := #str, IN2 := #value_0);
   #str := CONCAT_STRING(IN1 := #str, IN2 := '$t');
   #str := CONCAT_STRING(IN1 := #str, IN2 := #value_1);
   #str := CONCAT_STRING(IN1 := #str, IN2 := '$t');
   #str := CONCAT_STRING(IN1 := #str, IN2 := #value_2);

   "logger._log"(level := "LoggerLevels".INFO,
                 msg := #str
   );
END_FUNCTION

FUNCTION "logger.critical_3" : Void   // FC21, SCL
{ S7_Optimized_Access := 'TRUE' }
VERSION : 0.1
   VAR_INPUT
      msg : String;   // message for logging
      value_0 : String;   // additional value 0
      value_1 : String;   // additional value 1
      value_2 : String;   // additional value 2
   END_VAR
   VAR_TEMP
      str : String;
   END_VAR
BEGIN
   if "logger".config_in_block.level > "LoggerLevels".CRITICAL THEN
       return;
   END_IF;

   #str := '';
   #str := CONCAT_STRING(IN1 := #str, IN2 := #msg);
   #str := CONCAT_STRING(IN1 := #str, IN2 := '$t');
   #str := CONCAT_STRING(IN1 := #str, IN2 := #value_0);
   #str := CONCAT_STRING(IN1 := #str, IN2 := '$t');
   #str := CONCAT_STRING(IN1 := #str, IN2 := #value_1);
   #str := CONCAT_STRING(IN1 := #str, IN2 := '$t');
   #str := CONCAT_STRING(IN1 := #str, IN2 := #value_2);

   "logger._log"(level := "LoggerLevels".CRITICAL,
                 msg := #str
   );
END_FUNCTION

FUNCTION "logger.warning_3" : Void   // FC22, SCL
{ S7_Optimized_Access := 'TRUE' }
VERSION : 0.1
   VAR_INPUT
      msg : String;   // message for logging
      value_0 : String;   // additional value 0
      value_1 : String;   // additional value 1
      value_2 : String;   // additional value 2
   END_VAR
   VAR_TEMP
      str : String;
   END_VAR
BEGIN
   if "logger".config_in_block.level > "LoggerLevels".WARNING THEN
       return;
   END_IF;

   #str := '';
   #str := CONCAT_STRING(IN1 := #str, IN2 := #msg);
   #str := CONCAT_STRING(IN1 := #str, IN2 := '$t');
   #str := CONCAT_STRING(IN1 := #str, IN2 := #value_0);
   #str := CONCAT_STRING(IN1 := #str, IN2 := '$t');
   #str := CONCAT_STRING(IN1 := #str, IN2 := #value_1);
   #str := CONCAT_STRING(IN1 := #str, IN2 := '$t');
   #str := CONCAT_STRING(IN1 := #str, IN2 := #value_2);

   "logger._log"(level := "LoggerLevels".WARNING,
                 msg := #str
   );
END_FUNCTION